GLOBALCONSTANTS AID_TYPE (* Object type attribute id *)
  (* Standard: 61499-1; Description: Copyright (c) 2023 HR Agrartechnik GmbH This program and the accompanying materials are made available under the terms of the Eclipse Public License 2.0 which is available at https://www.eclipse.org/legal/epl-2.0/ SPDX-License-Identifier: EPL-2.0 *)
  (* Version 1.0, 2026-06-20, Franz Höpfinger, HR Agrartechnik GmbH *)
  PACKAGE isobus::UT::Q::const::AID;
  VAR_GLOBAL CONSTANT
    OBJ_TYPE : USINT := USINT#0; (* 0: AID_TYPE_OBJ_TYPE - Object Type identifier. *)
  END_VAR
END_GLOBALCONSTANTS
